(* CODESYS project Utility_functions.export

Project tree, tasks and I/O mapping:
  Utility_functions/
    function block Value_Clamp [ST]
*)

// Utility_functions/Value_Clamp
FUNCTION_BLOCK Value_Clamp
// clamp the input value between first value and second value
VAR_INPUT
	Current : REAL;
	First_Value : REAL;
	Second_value : REAL;
END_VAR
VAR_OUTPUT
	newV : REAL;
END_VAR
VAR
END_VAR

newV := Current;
IF First_Value < Second_value THEN
	IF Current < First_Value THEN
		newV := First_Value;
	END_IF
	IF Current > Second_value THEN
		newV := Second_value;
	END_IF
ELSIF First_Value > Second_value THEN
	IF Current > First_Value THEN
		newV := First_Value;
	END_IF
	IF Current < Second_value THEN
		newV := Second_value;
	END_IF
END_IF
// not going to deal the situation of first value equal to second value

END_FUNCTION_BLOCK
